PROGRAM Vision_Step
VAR
	Always_ON		:	BOOL	:=TRUE;	//상시ON
	Always_OFF		:	BOOL	:=FALSE;//상시OFF

	TEST01: BOOL;
	Test0002: INT;
	Data_Copy : R_TRIG;

END_VAR
VAR // added by the converter: edge detectors and wires of the graphical bodies
    _rt1, _rt2 : R_TRIG;
    _w1, _w2, _w3, _w4, _w5 : BOOL;
END_VAR

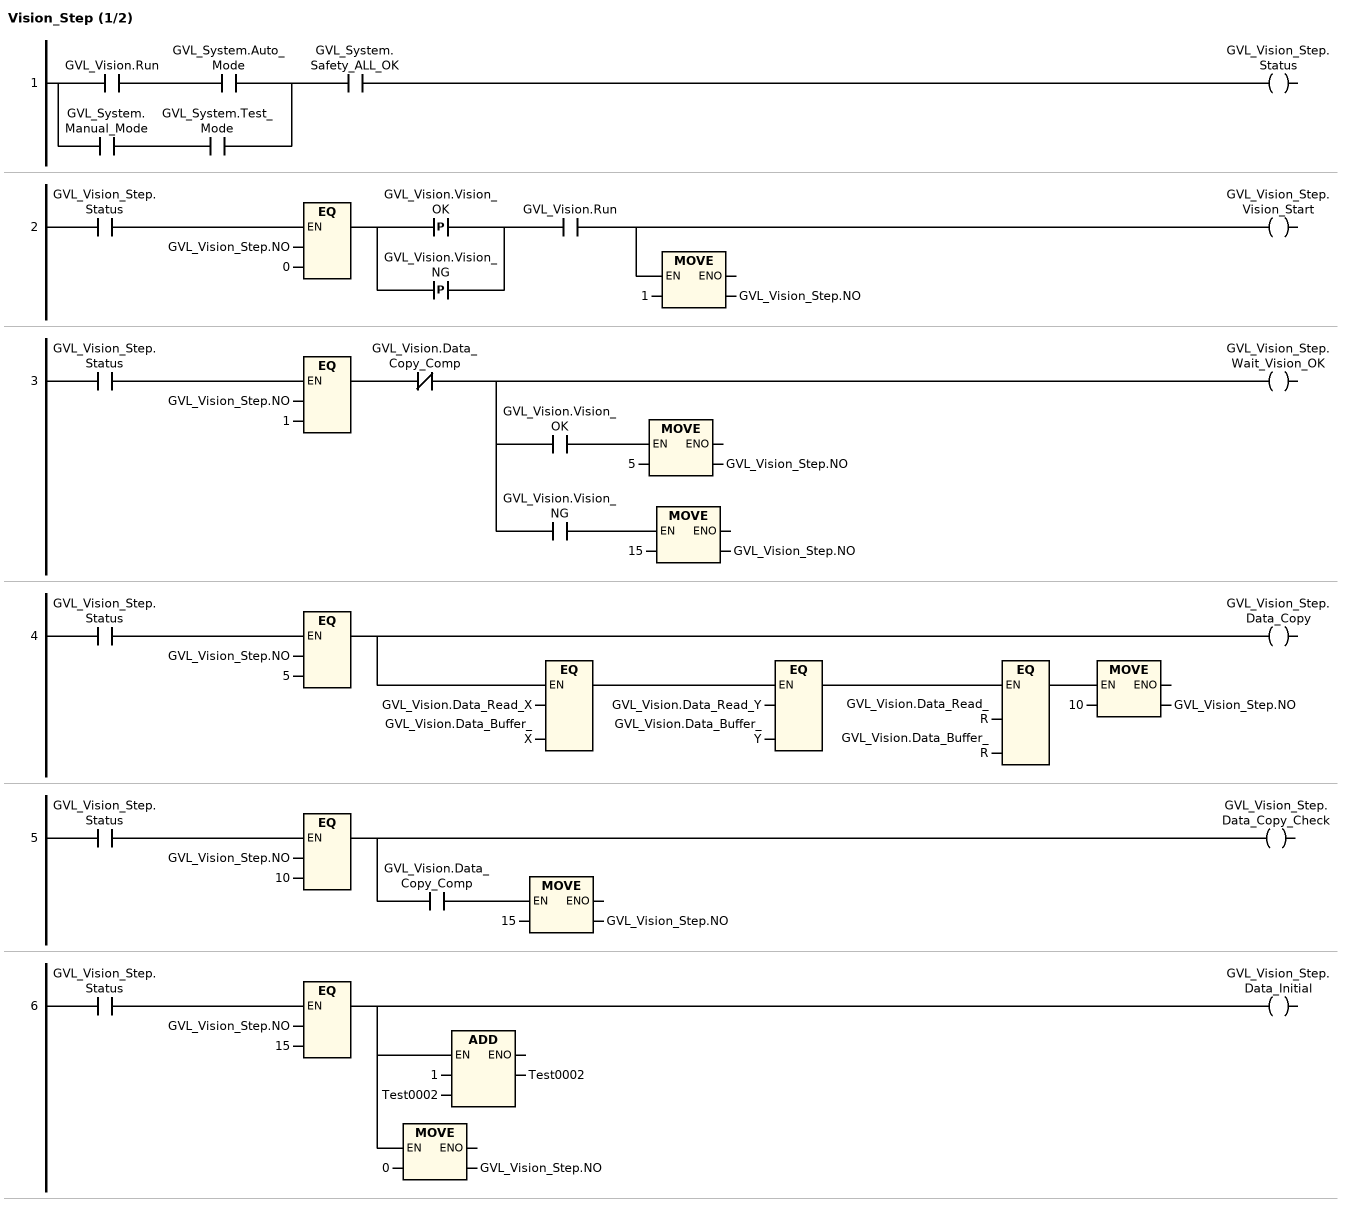
// NETWORK 1
GVL_Vision_Step.Status := (GVL_Vision.Run AND GVL_System.Auto_Mode OR GVL_System.Manual_Mode AND GVL_System.Test_Mode) AND GVL_System.Safety_ALL_OK;

// NETWORK 2
_rt1(CLK := GVL_Vision.Vision_OK);
_rt2(CLK := GVL_Vision.Vision_NG);
_w1 := (GVL_Vision_Step.Status AND GVL_Vision_Step.NO = 0) AND (_rt1.Q OR _rt2.Q) AND GVL_Vision.Run;
GVL_Vision_Step.Vision_Start := _w1;
IF _w1 THEN GVL_Vision_Step.NO := 1; END_IF

// NETWORK 3
_w2 := (GVL_Vision_Step.Status AND GVL_Vision_Step.NO = 1) AND NOT GVL_Vision.Data_Copy_Comp;
GVL_Vision_Step.Wait_Vision_OK := _w2;
IF _w2 AND GVL_Vision.Vision_OK THEN GVL_Vision_Step.NO := 5; END_IF
IF _w2 AND GVL_Vision.Vision_NG THEN GVL_Vision_Step.NO := 15; END_IF

// NETWORK 4
_w3 := GVL_Vision_Step.Status AND GVL_Vision_Step.NO = 5;
GVL_Vision_Step.Data_Copy := _w3;
IF _w3 AND GVL_Vision.Data_Read_X = GVL_Vision.Data_Buffer_X AND GVL_Vision.Data_Read_Y = GVL_Vision.Data_Buffer_Y AND GVL_Vision.Data_Read_R = GVL_Vision.Data_Buffer_R THEN
    GVL_Vision_Step.NO := 10;
END_IF

// NETWORK 5
_w4 := GVL_Vision_Step.Status AND GVL_Vision_Step.NO = 10;
GVL_Vision_Step.Data_Copy_Check := _w4;
IF _w4 AND GVL_Vision.Data_Copy_Comp THEN GVL_Vision_Step.NO := 15; END_IF

// NETWORK 6
_w5 := GVL_Vision_Step.Status AND GVL_Vision_Step.NO = 15;
GVL_Vision_Step.Data_Initial := _w5;
IF _w5 THEN Test0002 := 1 + Test0002; END_IF
IF _w5 THEN GVL_Vision_Step.NO := 0; END_IF

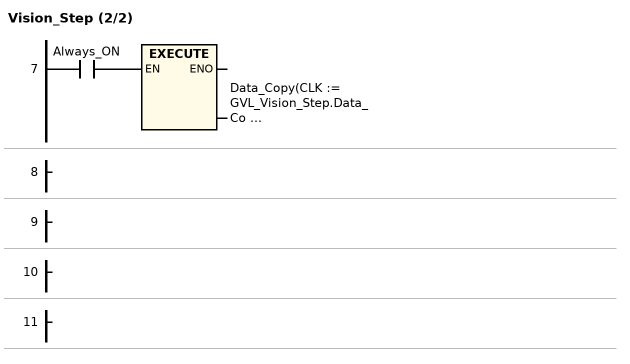
// NETWORK 7
IF Always_ON THEN
    Data_Copy(CLK := GVL_Vision_Step.Data_Copy);
    
    IF DATA_Copy.Q THEN
    GVL_Vision.Data_Buffer_X := GVL_Vision.Data_Read_X ;
    GVL_Vision.Data_Buffer_Y := GVL_Vision.Data_Read_Y ;
    GVL_Vision.Data_Buffer_R := GVL_Vision.Data_Read_R ;
    GVL_Vision.Data_Copy_Comp := 1 ;	
    END_IF
END_IF

// NETWORK 8

// NETWORK 9

// NETWORK 10

// NETWORK 11

END_PROGRAM

(* stored: Version 1.1.0.1, ProductVersion 3.1.4024.15
   POU Vision_Step: Id {e5cc5a74-cc08-4b0c-932f-421998a8f656}, SpecialFunc None *)
